# EPICS substitutions: streamApp/pluginDb/pluginROI.substitutions
#
# pluginROI.substitutions
#

file NDROI.template
{
	{
    PORT            = "ROI\$(N)",
    P               = "$(CAM):",
	R				= "$(PORT):",
    ADDR            = "\$(ADDR=0)",
    TIMEOUT         = "\$(TIMEOUT=1)",
    NDARRAY_PORT    = "\$(PLUGIN_SRC)",
    NDARRAY_ADDR    = "\$(NDARRAY_ADDR=0)",
	}
}
